TYPE InputBase_8311D824 :
STRUCT
END_STRUCT
END_TYPE

(* stored: Version 1.2.0.0, ProductVersion 3.1.4024.9
   DUT InputBase_8311D824: Id {d9e71b74-1b71-4b1c-bde2-f3369988b26f} *)
